// TIA Portal V17 export
// export: Created 2024-08-29T18:23:45.0401551Z, ExportSetting WithDefaults, DisplayName Totally Integrated Automation Portal, DisplayVersion V17 Update 7, DisplayName TIA Portal Openness, DisplayVersion V17 Update 7, DisplayName TIA Portal Version Control Interface, DisplayVersion V17, DisplayName SINAMICS Startdrive Advanced, DisplayVersion V17 SP2, DisplayName SINAMICS Startdrive G110M, G120, G120C, G120D, G120P, G115D, DisplayVersion V17 SP2, DisplayName SINAMICS Startdrive G130, G150, S120, S150, SINAMICS MV, S210, DisplayVersion V17 SP2, DisplayName STEP 7 Professional, DisplayVersion V17 Update 7, DisplayName STEP 7 Safety, DisplayVersion V17 Update 6, DisplayName WinCC Advanced / Unified PC, DisplayVersion V17 Update 7
DATA_BLOCK "DB_PrinterReference"   // DB33
{ S7_Optimized_Access := 'TRUE' }
VERSION : 0.1
// stored: AutoNumber true, DBAccessibleFromOPCUA true, DBAccessibleFromWebserver true, IsOnlyStoredInLoadMemory false, IsRetainMemResEnabled false, IsWriteProtectedInAS false, MemoryReserve 100
   VAR
      reference : Array[0..32] of "udt_referenceMainInfo";
   END_VAR
BEGIN
   reference[0..32].id := 0;
   reference[0..32].description := '';
   reference[0..32].partNumber := '';
   reference[0..32].rev := '';
   reference[0..32].customerNumber := '';
   reference[0..32].vpps := '';
   reference[0..32].locationCode := '';
   reference[0..32].dataIdentifier := '';
   reference[0..32].duns := '';
END_DATA_BLOCK
